PROGRAM PGR_Test
VAR
END_VAR

END_PROGRAM

(* stored: Version 1.1.0.1, ProductVersion 3.1.4024.12
   POU PGR_Test: Id {84d485d7-dc6d-4f01-863b-381f548c2345}, SpecialFunc None *)
